FUNCTION_BLOCK PUBLIC ABSTRACT TcoTaskedService EXTENDS TcoCore.TcoTask
VAR
	
END_VAR

(*~
	<docu>
		<summary>
			Main method of the sequener. Custom code needs to be placed here. The sequencer is executed by call of **Instance.Run()** method.
			This method is abstract, and it must be overridden in derived block.
		</summary>
	</docu>
~*)
METHOD PROTECTED ABSTRACT Main : BOOL
END_METHOD

(*~
	<docu>
		<summary>
			<para>
				Ensures calling the Open(), Main() and Close() methods in the desired order.
				This method is final, so it cannot be overloaded. The **Instance.Run()** needs to be called cyclically inside the appropriate context.
			</para>
		</summary>			
	</docu>	
~*)
METHOD PUBLIC FINAL Run
VAR
    _message : STRING;
END_VAR
IF (THIS^.Execute()) THEN
    THIS^.Main();    
END_IF;
END_METHOD

PROPERTY Task : REFERENCE TO TcoTask
GET
Task REF= THIS^;
END_GET
END_PROPERTY

END_FUNCTION_BLOCK

(* stored: Version 1.1.0.1, ProductVersion 3.1.4024.9
   POU TcoTaskedService: Id {204f6525-deb4-48a5-ab6d-4e0c7c871eb4}, SpecialFunc None
   Method Main: Id {cc5b8a36-a081-4438-80ce-668a9dfebbe4}
   Method Run: Id {3909f63a-de90-44dc-9203-0a4aa4366df2}
   Property Task: Id {31dc550d-fc4c-4312-b06a-80f3f9ff5603}
   Get Get: Id {26cb66eb-7f7f-4986-99db-29f80495fea7} *)
